FUNCTION_BLOCK FB_MockConfigProvider IMPLEMENTS I_GantryConfigProvider
VAR
    _MockConfig : ST_GantryXYZ_Config;
END_VAR

PROPERTY Config : ST_GantryXYZ_Config
GET
Config := _MockConfig;
END_GET
SET
_MockConfig := Config;
END_SET
END_PROPERTY

END_FUNCTION_BLOCK

(* stored: Version 1.1.0.1, ProductVersion 3.1.4024.15
   POU FB_MockConfigProvider: Id {1cf22c00-32b1-4334-b0ba-bb0033a9fe6a}, SpecialFunc None
   Property Config: Id {98ba9e04-c6dd-4bd0-953b-b00b87da8f4b}
   Get Get: Id {a7ec6669-d8cc-485f-ad66-71b6c5dd4e2e}
   Set Set: Id {7aa55b37-d946-42cb-bdab-7d5120bef258} *)
